// TIA Portal V19 export
TYPE "LEXCHANGETRAY_typeRoller_recieve_interface_B2"
// stored: Access Published
   STRUCT
      logistics : "LEXCHANGETRAY_typeRoller_toLogisticsRecieve_B2";
      workStationRoller : "LEXCHANGETRAY_typeRoller_toWorkstationRecieve_B2";
   END_STRUCT;
END_TYPE
